(* PLC project BlogProject.project, CODESYS CODESYS V3.5 SP14 Patch 3 *)
(* stored: creationDateTime 2021-10-07T21:07:10.7572103, modificationDateTime 2021-10-07T20:40:20.1109198 *)

FUNCTION_BLOCK mcNoEvent IMPLEMENTS itfEvent

            
          

METHOD getEvent : BOOL
                  getEvent:=true;
                
END_METHOD
END_FUNCTION_BLOCK
